# EPICS substitutions: examplesTop/ndsex1App/Db/Timestamping.substitutions
file "nds3_Timestamping.template" {
pattern
{
    BOARDTYPE,
    BOARDTYPEIDX,
    CBS1,
    CBS2,
    STATEMACHINE_PARENT,
    STATEMACHINE_NAME,
    TIMESTAMPING_NAME,
}

{
    "B",
    "0",
    "TEST",
    "FCT0",
    "Timestamping-",
    "StateMachine"
    "Timestamping",
}

}
